(* PLC project Tc3_EventLogger.FB_TcSourceInfo_Clear Demo, tc3-libraries-kb TwinCAT 3.1 *)
(* stored: creationDateTime 2026-05-11T01:00:00, modificationDateTime 2026-05-11T01:00:00 *)

PROGRAM P_Demo_FB_TcSourceInfo_Clear
  VAR
    fbTcSourceInfo : FB_TcSourceInfo;  (* Tc3_EventLogger.FB_TcSourceInfo 实例 *)
  END_VAR

            // ============================================================
// Tc3_EventLogger.FB_TcSourceInfo.Clear 演示程序（OO 方法）
// ============================================================
// 验证步骤：
//   1. 引用 Tc3_EventLogger（及依赖类型所在库 Tc2_System 等）
//   2. 编译 + 登录
//   3. 按 doc.md 给 arg_* 赋值
//   4. 在线监视 out_* / io_* 输出
// ============================================================

fbTcSourceInfo.Clear(

);

          
END_PROGRAM
